PROGRAM TestPrg
VAR
END_VAR

TC_EVENTS.ST_Warning.event1;

END_PROGRAM

(* stored: Version 1.1.0.1
   POU TestPrg: Id {180aa939-3755-4e05-bbd0-449d032be2e9}, SpecialFunc None *)
